{attribute 'qualified_only'}
{attribute 'strict'}
TYPE E_ReloadRoundBoxAction :
(
	Undefined := 0,
	ClampA_WareHouseA,
	ClampA_WareHouseB,
	ClampB_WareHouseA,
	ClampB_WareHouseB,
	A_WareHouseA_B_WareHouseA,
	A_WareHouseA_B_WareHouseB,
	A_WareHouseB_B_WareHouseA,
	A_WareHouseB_B_WareHouseB
);
END_TYPE

(* stored: Version 1.1.0.1, ProductVersion 3.1.4024.13
   DUT E_ReloadRoundBoxAction: Id {b38be6b1-240b-48c6-926b-de3882876ffd} *)
